{attribute addProperty BoxType "EL1918-0000-0016"}
{attribute addProperty Id "FSOEAT %Q*FSOE_F2812FEE486"}
{attribute addProperty CRC "1855391509"}
{attribute addProperty SizeInBites "48"}
{attribute addProperty SizeInBytes "6"}
TYPE FSoE_Outputs_6E970715 :
STRUCT
	{attribute addProperty Name "FSOE"}
	FSOE AT %Q* : FSOE_F2812FEE;
END_STRUCT
END_TYPE

(* stored: Version 1.2.0.0, ProductVersion 3.1.4024.9
   DUT FSoE_Outputs_6E970715: Id {5fdb79f9-b802-4415-8886-c7a7c4f7e1e8} *)
